{attribute 'GeneratedUsingTerminal: EJ2502-0000-0023'}
{attribute addProperty BoxType "EJ2502-0000-0023"}
{attribute addProperty Id "PWM_Outputs_Channel_1AT %Q*PWM_Outputs_Channel_4C6289CD2PWM_Outputs_Channel_2AT %Q*PWM_Outputs_Channel_4C6289CD2WcStateAT %I*WcState_0B2B16F91InfoDataAT %I*InfoData_94A18F5E2"}
{attribute addProperty CRC "2304954225"}
{attribute addProperty Size "7"}
TYPE EJ2502_8962CF71 EXTENDS EtcSlaveTerminalBase_947E5A46 :
STRUCT
	{attribute addProperty Name "PWM_Outputs_Channel_1"}
	PWM_Outputs_Channel_1 : PWM_Outputs_Channel_4C6289CD;
	{attribute addProperty Name "PWM_Outputs_Channel_2"}
	PWM_Outputs_Channel_2 : PWM_Outputs_Channel_4C6289CD;
	{attribute addProperty Name "WcState"}
	WcState : WcState_0B2B16F9;
	{attribute addProperty Name "InfoData"}
	InfoData : InfoData_94A18F5E;
END_STRUCT
END_TYPE

(* stored: Version 1.2.0.0, ProductVersion 3.1.4024.9
   DUT EJ2502_8962CF71: Id {ca03e779-bac7-4b37-978f-86191bc76ef0} *)
